(* CODESYS project CUS-1974

Project tree, tasks and I/O mapping:
  Device : CODESYS Control for Raspberry Pi MC SL, CODESYS GmbH, order no. 2302000009, version 4.9.0.0
    application Application
      libraries: Standard, 3.5.18.0 (System)
      task MainTask (cyclic, interval t#4ms, priority 1) calls PLC_PRG
      program PLC_PRG [ST]
    Camera device
      <Empty>
    GPIOs_A_B : GPIOs A/B, 3S - Smart Software Solutions GmbH, version 4.9.0.0
        unmapped channels: digital inputs (GPIO0..GPIO31), digital outputs (GPIO0..GPIO31)
    I²C
    Onewire
    SoftMotion General Axis Pool
    SPI
*)

// Device/Application/PLC_PRG
PROGRAM PLC_PRG
VAR
	bChange : BOOL;
	bChange2 : BOOL;
	bChange3 : BOOL;
END_VAR

END_PROGRAM
